INTERFACE I_DataChannelRecv

METHOD GetData : BOOL
VAR_INPUT
	udiDataSize				: UDINT;
	pData					: POINTER TO BYTE;
END_VAR
END_METHOD

PROPERTY Busy : BOOL
GET
END_GET
END_PROPERTY

METHOD InitChannel : BOOL
VAR_INPUT
	udiDataSize					: UDINT;
	pInputData					: POINTER TO BYTE;
END_VAR
END_METHOD

PROPERTY DataSize : UDINT
GET
END_GET
END_PROPERTY

PROPERTY Error : INT
GET
END_GET
SET
END_SET
END_PROPERTY

END_INTERFACE

(* stored: Version 1.1.0.1, ProductVersion 3.1.0.24
   Itf I_DataChannelRecv: Id {0ef3c332-df02-4c0e-a934-81440cf192b5}
   Method GetData: Id {0909c4e5-8eac-4a33-877d-aa68fb131bf9}
   Property Busy: Id {0bbdc364-9cb3-48c7-bd3a-63758dd4a48a}
   Get Get: Id {cc3ebaf1-2da2-400f-9505-71de6d1bfc8c}
   Method InitChannel: Id {6149d0cb-e235-4d0b-8512-d044c47a954f}
   Property DataSize: Id {c2ef2a79-0d85-49c8-b2aa-85709a86d043}
   Get Get: Id {9e147ab5-cd4a-4bfd-8353-bbdb149c928d}
   Property Error: Id {f385048f-5343-48a6-85d5-3e6607226846}
   Get Get: Id {35851331-4966-4720-8ec9-b3b441fd1bb5}
   Set Set: Id {504f7d93-bccb-4cef-8085-cc9481eeab7b} *)
